// TwinCAT 3 PLC project FileUpload
// ProgramVersion: 3.1.0.5
// libraries:
//   Tc2_FTP,newest,Beckhoff Automation GmbH
//   Tc2_Standard,newest,Beckhoff Automation GmbH
//   Tc2_System,newest,Beckhoff Automation GmbH
//   Tc3_Module,newest,Beckhoff Automation GmbH
// project tree:
//   / PlcTask.TcTTO
//   POUs/ MAIN.TcPOU
// real-time tasks:
//   TASK PlcTask: cycle T#10ms, priority 20, ADS port 350

CONFIGURATION FileUpload
    RESOURCE PLC ON TwinCAT3
        TASK PlcTask(INTERVAL := T#10ms, PRIORITY := 20);
        PROGRAM MAIN WITH PlcTask : MAIN;
    END_RESOURCE
END_CONFIGURATION

// ---- POUs/MAIN.TcPOU
PROGRAM MAIN
VAR
	FB_FTPFileUpload1	: FB_FTP_FileUploadEx;
	startstop			: BOOL;
	busy				: BOOL;
	err					: BOOL;
	errid				: UDINT;
	progress			: UDINT;
END_VAR

FB_FTPFileUpload1(
	sNetID:= ,
	sHost:= '172.17.36.148',
	nPort:= DEFAULT_FTP_PORT,
	sUsername:= 'TestUser',
	sPassword:= 'TestPwd123',
	sSrcFile:= '\Program Files\TestFile1.txt',
	sDesFile:= '\TestFolder\File1.txt',
	bExecute:= startstop,
	tTimeout:= T#15s,
	bBusy=> busy,
	bError=> err,
	nErrId=> errid,
	nProgress=> progress);

END_PROGRAM
